(* Logix 5000 project; controller p65 vendor 1 type 14 code 85 rev 20.11; software revision 20.01; part 6 of 7 *)
(* tags used below, declared in another part *)
   DCMicroGridisInOperation : ALIAS FOR DINT00_23.8;
   DCMicroGridisSimulating : ALIAS FOR DINT00_23.10;
   Load03accountBalance : ALIAS FOR REAL00_63;
   Load03accountDepositRate : ALIAS FOR REAL00_64;
   Load03Bclose : ALIAS FOR Local:3:O.Data.7;
   Load03BcloseHILS : ALIAS FOR plc1_local_6[0].7;
   Load03BcloseProxy : ALIAS FOR DINT00_25.11;
   Load03BintReqClose : ALIAS FOR DINT00_25.12;
   Load03BisClosed : ALIAS FOR DINT00_25.13;
   Load03BisOpen : ALIAS FOR DINT00_25.14;
   Load03BreqClose : ALIAS FOR DINT00_25.15;
   Load03BreqOpen : ALIAS FOR DINT00_25.16;
   Load03commandChanged : ALIAS FOR DINT00_25.17;
   Load03commandChangedTimer : ALIAS FOR CLTIMER00_23;
   Load03current : ALIAS FOR REAL00_65;
   Load03currentHILS : ALIAS FOR plc1_local_2[7];
   Load03currentRaw : ALIAS FOR Local:2:I.Ch4Data;
   Load03deadband : ALIAS FOR REAL00_66;
   Load03depositTimer : ALIAS FOR CLTIMER00_24;
   Load03DisconnectPowerEventFail : ALIAS FOR DINT00_25.18;
   Load03DisconnectPowerEventSuccess : ALIAS FOR DINT00_25.19;
   Load03DisconnectPowerFailTimer : ALIAS FOR CLTIMER00_25;
   Load03DisconnectPowerInProcess : ALIAS FOR DINT00_25.20;
   Load03DisconnectPowerMsg : ALIAS FOR MESSAGE00_5;
   Load03DisconnectPowerSuccessTimer : ALIAS FOR CLTIMER00_26;
   Load03failedToConnect : ALIAS FOR DINT00_25.21;
   Load03failedToDisconnect : ALIAS FOR DINT00_25.22;
   Load03fundsAvailable : ALIAS FOR DINT00_25.23;
   Load03incrementToAdd : ALIAS FOR REAL00_67;
   Load03incrementToSubtract : ALIAS FOR REAL00_68;
   Load03intReqConnect : ALIAS FOR DINT00_25.24;
   Load03isConnected : ALIAS FOR DINT00_25.25;
   Load03isDisconnected : ALIAS FOR DINT00_25.26;
   Load03minBalance : ALIAS FOR REAL00_70;
   Load03minBalanceToReconnect : ALIAS FOR REAL00_71;
   Load03minTime : ALIAS FOR REAL00_72;
   Load03powerRate : ALIAS FOR REAL00_73;
   Load03powerRateMax : REAL;
   Load03PurchasePowerEventFail : ALIAS FOR DINT00_25.27;
   Load03PurchasePowerEventSuccess : ALIAS FOR DINT00_25.28;
   Load03PurchasePowerFailTimer : ALIAS FOR CLTIMER00_27;
   Load03PurchasePowerInProcess : ALIAS FOR DINT00_25.29;
   Load03PurchasePowerMsg : ALIAS FOR MESSAGE00_6;
   Load03PurchasePowerSuccessTimer : ALIAS FOR CLTIMER00_28;
   Load03reqConnect : ALIAS FOR DINT00_25.30;
   Load03reqDisconnect : ALIAS FOR DINT00_25.31;
   Load03runningOut : ALIAS FOR DINT00_26.0;
   Load03spendingRate : ALIAS FOR REAL00_74;
   Load03timeRemaining : ALIAS FOR REAL00_75;
   Load03usageTimer : ALIAS FOR CLTIMER00_29;
   Load04accountBalance : ALIAS FOR REAL00_76;
   Load04accountDepositRate : ALIAS FOR REAL00_77;
   Load04Bclose : ALIAS FOR Local:3:O.Data.8;
   Load04BcloseHILS : ALIAS FOR plc1_local_6[0].8;
   Load04BcloseProxy : ALIAS FOR DINT00_26.1;
   Load04BintReqClose : ALIAS FOR DINT00_26.2;
   Load04BisClosed : ALIAS FOR DINT00_26.3;
   Load04BisOpen : ALIAS FOR DINT00_26.4;
   Load04BreqClose : ALIAS FOR DINT00_26.5;
   Load04BreqOpen : ALIAS FOR DINT00_26.6;
   Load04commandChanged : ALIAS FOR DINT00_26.7;
   Load04commandChangedTimer : ALIAS FOR CLTIMER00_30;
   Load04current : ALIAS FOR REAL00_78;
   Load04currentHILS : ALIAS FOR plc1_local_2[8];
   Load04currentRaw : ALIAS FOR Local:2:I.Ch5Data;
   Load04deadband : ALIAS FOR REAL00_79;
   Load04depositTimer : ALIAS FOR CLTIMER00_31;
   Load04DisconnectPowerEventFail : ALIAS FOR DINT00_26.8;
   Load04DisconnectPowerEventSuccess : ALIAS FOR DINT00_26.9;
   Load04DisconnectPowerFailTimer : ALIAS FOR CLTIMER00_32;
   Load04DisconnectPowerInProcess : ALIAS FOR DINT00_26.10;
   Load04DisconnectPowerMsg : ALIAS FOR MESSAGE00_7;
   Load04DisconnectPowerSuccessTimer : ALIAS FOR CLTIMER00_33;
   Load04failedToConnect : ALIAS FOR DINT00_26.11;
   Load04failedToDisconnect : ALIAS FOR DINT00_26.12;
   Load04fundsAvailable : ALIAS FOR DINT00_26.13;
   Load04incrementToAdd : ALIAS FOR REAL00_80;
   Load04incrementToSubtract : ALIAS FOR REAL00_81;
   Load04intReqConnect : ALIAS FOR DINT00_26.14;
   Load04isConnected : ALIAS FOR DINT00_26.15;
   Load04isDisconnected : ALIAS FOR DINT00_26.16;
   Load04minBalance : ALIAS FOR REAL00_83;
   Load04minBalanceToReconnect : ALIAS FOR REAL00_84;
   Load04minTime : ALIAS FOR REAL00_85;
   Load04powerRate : ALIAS FOR REAL00_86;
   Load04powerRateMax : REAL;
   Load04PurchasePowerEventFail : ALIAS FOR DINT00_26.17;
   Load04PurchasePowerEventSuccess : ALIAS FOR DINT00_26.18;
   Load04PurchasePowerFailTimer : ALIAS FOR CLTIMER00_34;
   Load04PurchasePowerInProcess : ALIAS FOR DINT00_26.19;
   Load04PurchasePowerMsg : ALIAS FOR MESSAGE00_8;
   Load04PurchasePowerSuccessTimer : ALIAS FOR CLTIMER00_35;
   Load04reqConnect : ALIAS FOR DINT00_26.20;
   Load04reqDisconnect : ALIAS FOR DINT00_26.21;
   Load04runningOut : ALIAS FOR DINT00_26.22;
   Load04spendingRate : ALIAS FOR REAL00_87;
   Load04timeRemaining : ALIAS FOR REAL00_88;
   Load04usageTimer : ALIAS FOR CLTIMER00_36;
   Load05accountBalance : ALIAS FOR REAL00_89;
   Load05accountDepositRate : ALIAS FOR REAL00_90;
   Load05Bclose : ALIAS FOR Local:3:O.Data.9;
   Load05BcloseHILS : ALIAS FOR plc1_local_6[0].9;
   Load05BcloseProxy : ALIAS FOR DINT00_26.23;
   Load05BintReqClose : ALIAS FOR DINT00_26.24;
   Load05BisClosed : ALIAS FOR DINT00_26.25;
   Load05BisOpen : ALIAS FOR DINT00_26.26;
   Load05BreqClose : ALIAS FOR DINT00_26.27;
   Load05BreqOpen : ALIAS FOR DINT00_26.28;
   Load05commandChanged : ALIAS FOR DINT00_26.29;
   Load05commandChangedTimer : ALIAS FOR CLTIMER00_37;
   Load05current : ALIAS FOR REAL00_91;
   Load05currentHILS : ALIAS FOR plc1_local_2[9];
   Load05currentRaw : ALIAS FOR Local:2:I.Ch6Data;
   Load05deadband : ALIAS FOR REAL00_92;
   Load05depositTimer : ALIAS FOR CLTIMER00_38;
   Load05DisconnectPowerEventFail : ALIAS FOR DINT00_26.30;
   Load05DisconnectPowerEventSuccess : ALIAS FOR DINT00_26.31;
   Load05DisconnectPowerFailTimer : ALIAS FOR CLTIMER00_39;
   Load05DisconnectPowerInProcess : ALIAS FOR DINT00_27.0;
   Load05DisconnectPowerMsg : ALIAS FOR MESSAGE00_9;
   Load05DisconnectPowerSuccessTimer : ALIAS FOR CLTIMER00_40;
   Load05failedToConnect : ALIAS FOR DINT00_27.1;
   Load05failedToDisconnect : ALIAS FOR DINT00_27.2;
   Load05fundsAvailable : ALIAS FOR DINT00_27.3;
   Load05incrementToAdd : ALIAS FOR REAL00_93;
   Load05incrementToSubtract : ALIAS FOR REAL00_94;
   Load05intReqConnect : ALIAS FOR DINT00_27.4;
   Load05isConnected : ALIAS FOR DINT00_27.5;
   Load05isDisconnected : ALIAS FOR DINT00_27.6;
   Load05minBalance : ALIAS FOR REAL00_96;
   Load05minBalanceToReconnect : ALIAS FOR REAL00_97;
   Load05minTime : ALIAS FOR REAL00_98;
   Load05powerRate : ALIAS FOR REAL00_99;
   Load05powerRateMax : REAL;
   Load05PurchasePowerEventFail : ALIAS FOR DINT00_27.7;
   Load05PurchasePowerEventSuccess : ALIAS FOR DINT00_27.8;
   Load05PurchasePowerFailTimer : ALIAS FOR CLTIMER00_41;
   Load05PurchasePowerInProcess : ALIAS FOR DINT00_27.9;
   Load05PurchasePowerMsg : ALIAS FOR MESSAGE00_10;
   Load05PurchasePowerSuccessTimer : ALIAS FOR CLTIMER00_42;
   Load05reqConnect : ALIAS FOR DINT00_27.10;
   Load05reqDisconnect : ALIAS FOR DINT00_27.11;
   Load05runningOut : ALIAS FOR DINT00_27.12;
   Load05spendingRate : ALIAS FOR REAL00_100;
   Load05timeRemaining : ALIAS FOR REAL00_101;
   Load05usageTimer : ALIAS FOR CLTIMER00_43;
   LoadslowVoltage : ALIAS FOR DINT00_27.23;
   UsingAgents : BOOL;

PROGRAM Load03   (* main routine Load03 *)

ROUTINE Load03   (* ladder *)
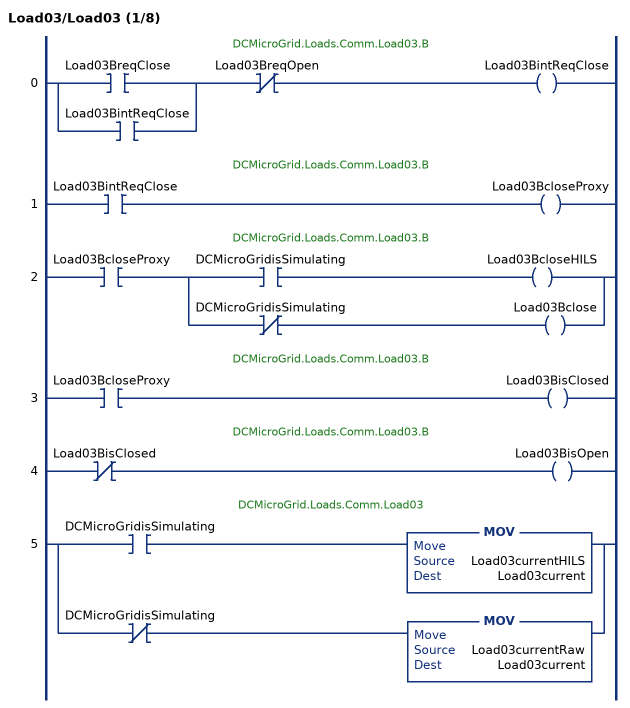
   // DCMicroGrid.Loads.Comm.Load03.B
   0: [XIC(Load03BreqClose) ,XIC(Load03BintReqClose) ]XIO(Load03BreqOpen)OTE(Load03BintReqClose);
   // DCMicroGrid.Loads.Comm.Load03.B
   1: XIC(Load03BintReqClose)OTE(Load03BcloseProxy);
   // DCMicroGrid.Loads.Comm.Load03.B
   2: XIC(Load03BcloseProxy)[XIC(DCMicroGridisSimulating) OTE(Load03BcloseHILS) ,XIO(DCMicroGridisSimulating) OTE(Load03Bclose) ];
   // DCMicroGrid.Loads.Comm.Load03.B
   3: XIC(Load03BcloseProxy)OTE(Load03BisClosed);
   // DCMicroGrid.Loads.Comm.Load03.B
   4: XIO(Load03BisClosed)OTE(Load03BisOpen);
   // DCMicroGrid.Loads.Comm.Load03
   5: [XIC(DCMicroGridisSimulating) MOV(Load03currentHILS,Load03current) ,XIO(DCMicroGridisSimulating) MOV(Load03currentRaw,Load03current) ];
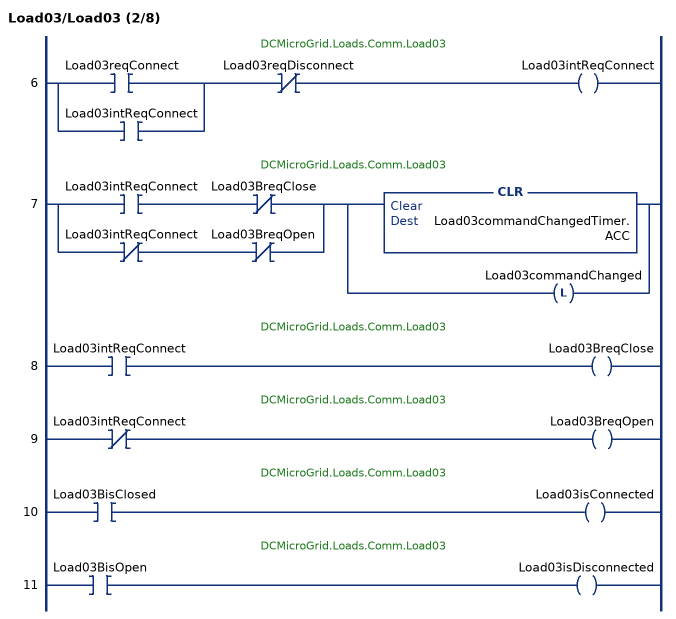
   // DCMicroGrid.Loads.Comm.Load03
   6: [XIC(Load03reqConnect) ,XIC(Load03intReqConnect) ]XIO(Load03reqDisconnect)OTE(Load03intReqConnect);
   // DCMicroGrid.Loads.Comm.Load03
   7: [XIC(Load03intReqConnect) XIO(Load03BreqClose) ,XIO(Load03intReqConnect) XIO(Load03BreqOpen) ][CLR(Load03commandChangedTimer.ACC) ,OTL(Load03commandChanged) ];
   // DCMicroGrid.Loads.Comm.Load03
   8: XIC(Load03intReqConnect)OTE(Load03BreqClose);
   // DCMicroGrid.Loads.Comm.Load03
   9: XIO(Load03intReqConnect)OTE(Load03BreqOpen);
   // DCMicroGrid.Loads.Comm.Load03
   10: XIC(Load03BisClosed)OTE(Load03isConnected);
   // DCMicroGrid.Loads.Comm.Load03
   11: XIC(Load03BisOpen)OTE(Load03isDisconnected);
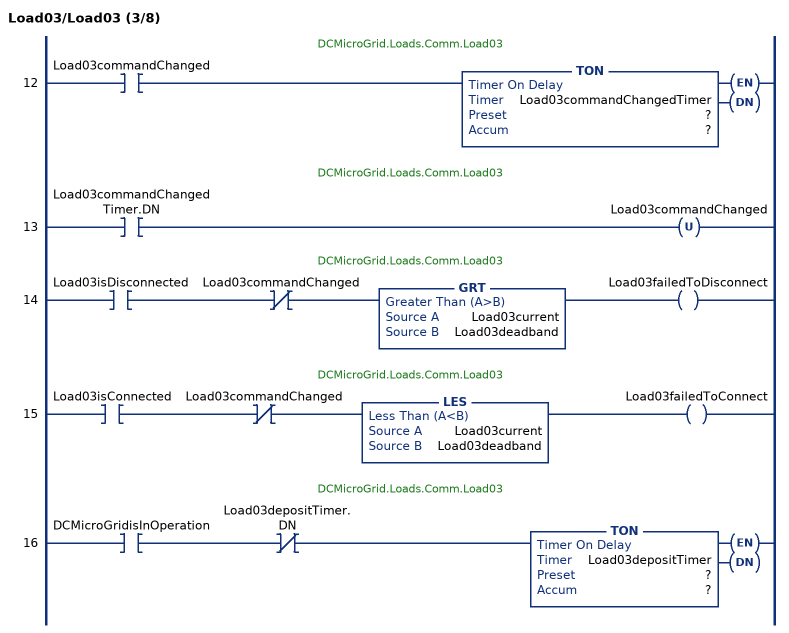
   // DCMicroGrid.Loads.Comm.Load03
   12: XIC(Load03commandChanged)TON(Load03commandChangedTimer,?,?);
   // DCMicroGrid.Loads.Comm.Load03
   13: XIC(Load03commandChangedTimer.DN)OTU(Load03commandChanged);
   // DCMicroGrid.Loads.Comm.Load03
   14: XIC(Load03isDisconnected)XIO(Load03commandChanged)GRT(Load03current,Load03deadband)OTE(Load03failedToDisconnect);
   // DCMicroGrid.Loads.Comm.Load03
   15: XIC(Load03isConnected)XIO(Load03commandChanged)LES(Load03current,Load03deadband)OTE(Load03failedToConnect);
   // DCMicroGrid.Loads.Comm.Load03
   16: XIC(DCMicroGridisInOperation)XIO(Load03depositTimer.DN)TON(Load03depositTimer,?,?);
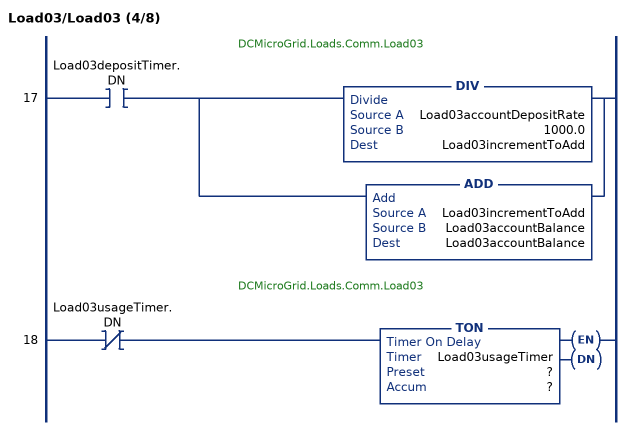
   // DCMicroGrid.Loads.Comm.Load03
   17: XIC(Load03depositTimer.DN)[DIV(Load03accountDepositRate,1000.0,Load03incrementToAdd) ,ADD(Load03incrementToAdd,Load03accountBalance,Load03accountBalance) ];
   // DCMicroGrid.Loads.Comm.Load03
   18: XIO(Load03usageTimer.DN)TON(Load03usageTimer,?,?);
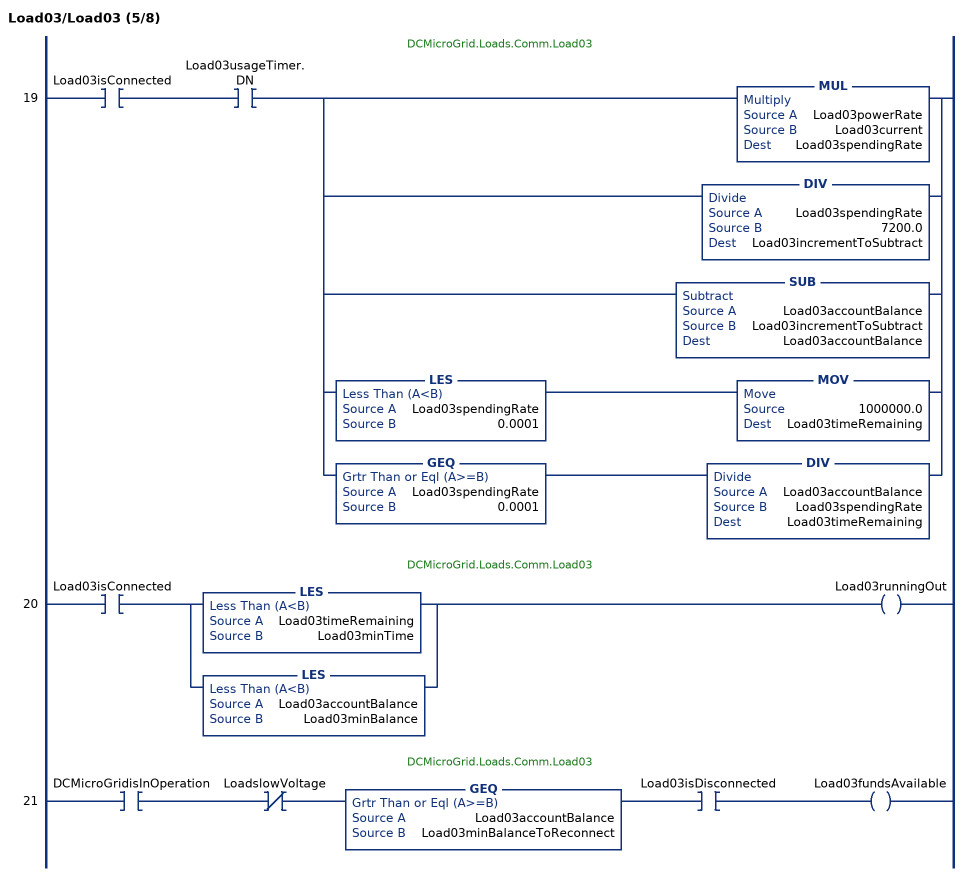
   // DCMicroGrid.Loads.Comm.Load03
   19: XIC(Load03isConnected)XIC(Load03usageTimer.DN)[MUL(Load03powerRate,Load03current,Load03spendingRate) ,DIV(Load03spendingRate,7200.0,Load03incrementToSubtract) ,SUB(Load03accountBalance,Load03incrementToSubtract,Load03accountBalance) ,[LES(Load03spendingRate,0.0001) MOV(1000000.0,Load03timeRemaining) ,GEQ(Load03spendingRate,0.0001) DIV(Load03accountBalance,Load03spendingRate,Load03timeRemaining) ] ];
   // DCMicroGrid.Loads.Comm.Load03
   20: XIC(Load03isConnected)[LES(Load03timeRemaining,Load03minTime) ,LES(Load03accountBalance,Load03minBalance) ]OTE(Load03runningOut);
   // DCMicroGrid.Loads.Comm.Load03
   21: XIC(DCMicroGridisInOperation)XIO(LoadslowVoltage)GEQ(Load03accountBalance,Load03minBalanceToReconnect)XIC(Load03isDisconnected)OTE(Load03fundsAvailable);
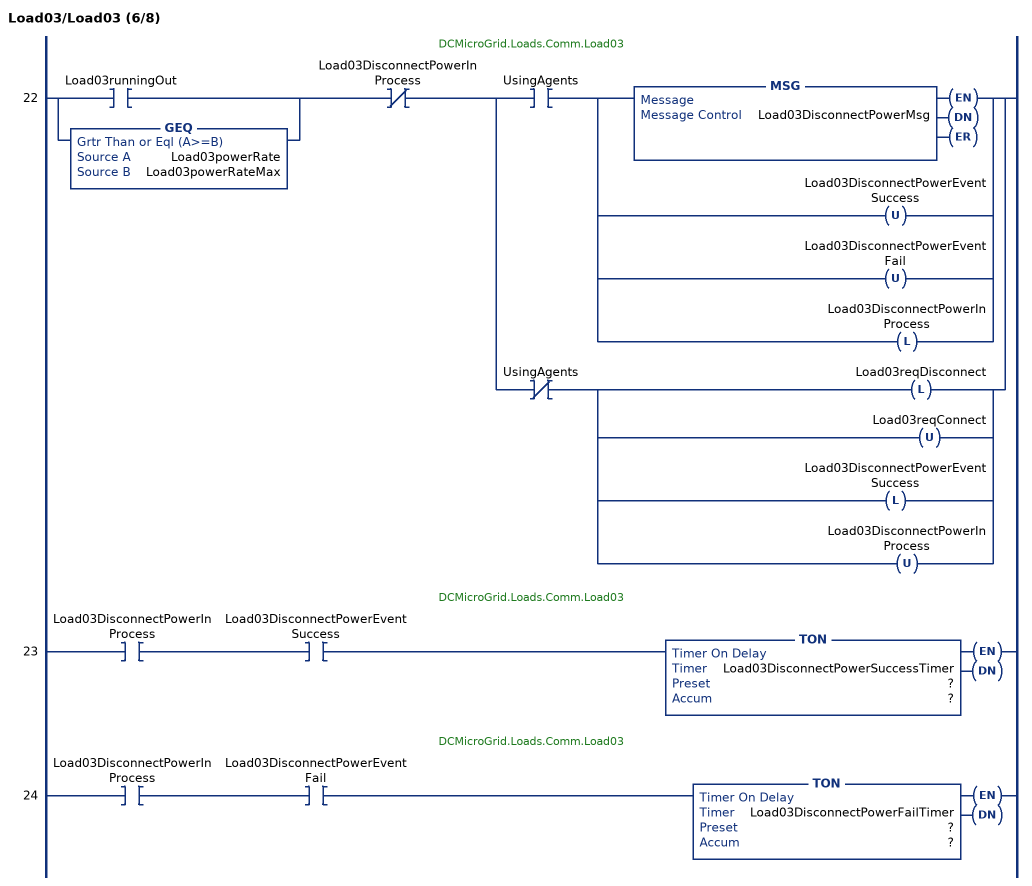
   // DCMicroGrid.Loads.Comm.Load03
   22: [XIC(Load03runningOut) ,GEQ(Load03powerRate,Load03powerRateMax) ]XIO(Load03DisconnectPowerInProcess)[XIC(UsingAgents) [MSG(Load03DisconnectPowerMsg) ,OTU(Load03DisconnectPowerEventSuccess) ,OTU(Load03DisconnectPowerEventFail) ,OTL(Load03DisconnectPowerInProcess) ] ,XIO(UsingAgents) [OTL(Load03reqDisconnect) ,OTU(Load03reqConnect) ,OTL(Load03DisconnectPowerEventSuccess) ,OTU(Load03DisconnectPowerInProcess) ] ];
   // DCMicroGrid.Loads.Comm.Load03
   23: XIC(Load03DisconnectPowerInProcess)XIC(Load03DisconnectPowerEventSuccess)TON(Load03DisconnectPowerSuccessTimer,?,?);
   // DCMicroGrid.Loads.Comm.Load03
   24: XIC(Load03DisconnectPowerInProcess)XIC(Load03DisconnectPowerEventFail)TON(Load03DisconnectPowerFailTimer,?,?);
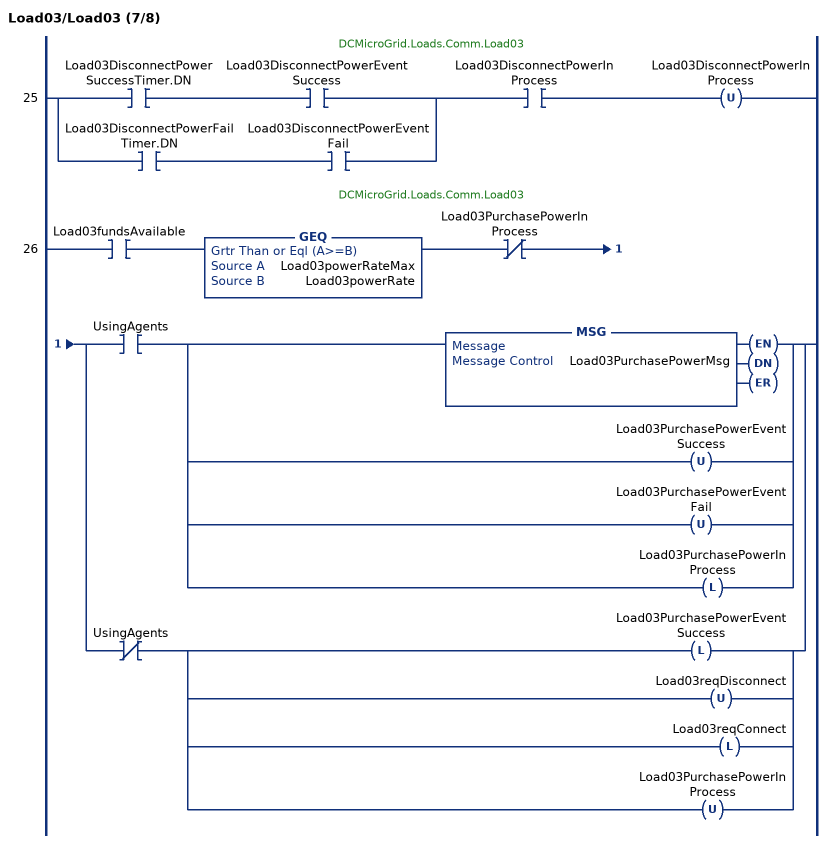
   // DCMicroGrid.Loads.Comm.Load03
   25: [XIC(Load03DisconnectPowerSuccessTimer.DN) XIC(Load03DisconnectPowerEventSuccess) ,XIC(Load03DisconnectPowerFailTimer.DN) XIC(Load03DisconnectPowerEventFail) ]XIC(Load03DisconnectPowerInProcess)OTU(Load03DisconnectPowerInProcess);
   // DCMicroGrid.Loads.Comm.Load03
   26: XIC(Load03fundsAvailable)GEQ(Load03powerRateMax,Load03powerRate)XIO(Load03PurchasePowerInProcess)[XIC(UsingAgents) [MSG(Load03PurchasePowerMsg) ,OTU(Load03PurchasePowerEventSuccess) ,OTU(Load03PurchasePowerEventFail) ,OTL(Load03PurchasePowerInProcess) ] ,XIO(UsingAgents) [OTL(Load03PurchasePowerEventSuccess) ,OTU(Load03reqDisconnect) ,OTL(Load03reqConnect) ,OTU(Load03PurchasePowerInProcess) ] ];
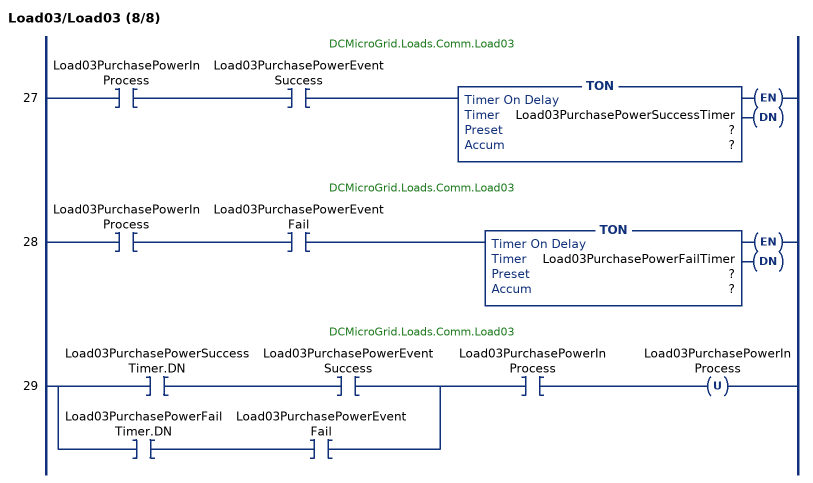
   // DCMicroGrid.Loads.Comm.Load03
   27: XIC(Load03PurchasePowerInProcess)XIC(Load03PurchasePowerEventSuccess)TON(Load03PurchasePowerSuccessTimer,?,?);
   // DCMicroGrid.Loads.Comm.Load03
   28: XIC(Load03PurchasePowerInProcess)XIC(Load03PurchasePowerEventFail)TON(Load03PurchasePowerFailTimer,?,?);
   // DCMicroGrid.Loads.Comm.Load03
   29: [XIC(Load03PurchasePowerSuccessTimer.DN) XIC(Load03PurchasePowerEventSuccess) ,XIC(Load03PurchasePowerFailTimer.DN) XIC(Load03PurchasePowerEventFail) ]XIC(Load03PurchasePowerInProcess)OTU(Load03PurchasePowerInProcess);
END_ROUTINE
END_PROGRAM

PROGRAM Load04   (* main routine Load04 *)

ROUTINE Load04   (* ladder *)
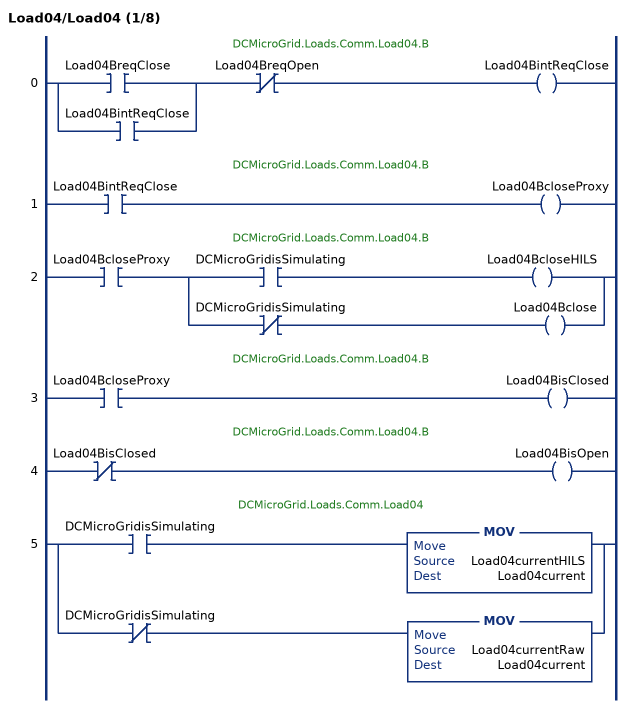
   // DCMicroGrid.Loads.Comm.Load04.B
   0: [XIC(Load04BreqClose) ,XIC(Load04BintReqClose) ]XIO(Load04BreqOpen)OTE(Load04BintReqClose);
   // DCMicroGrid.Loads.Comm.Load04.B
   1: XIC(Load04BintReqClose)OTE(Load04BcloseProxy);
   // DCMicroGrid.Loads.Comm.Load04.B
   2: XIC(Load04BcloseProxy)[XIC(DCMicroGridisSimulating) OTE(Load04BcloseHILS) ,XIO(DCMicroGridisSimulating) OTE(Load04Bclose) ];
   // DCMicroGrid.Loads.Comm.Load04.B
   3: XIC(Load04BcloseProxy)OTE(Load04BisClosed);
   // DCMicroGrid.Loads.Comm.Load04.B
   4: XIO(Load04BisClosed)OTE(Load04BisOpen);
   // DCMicroGrid.Loads.Comm.Load04
   5: [XIC(DCMicroGridisSimulating) MOV(Load04currentHILS,Load04current) ,XIO(DCMicroGridisSimulating) MOV(Load04currentRaw,Load04current) ];
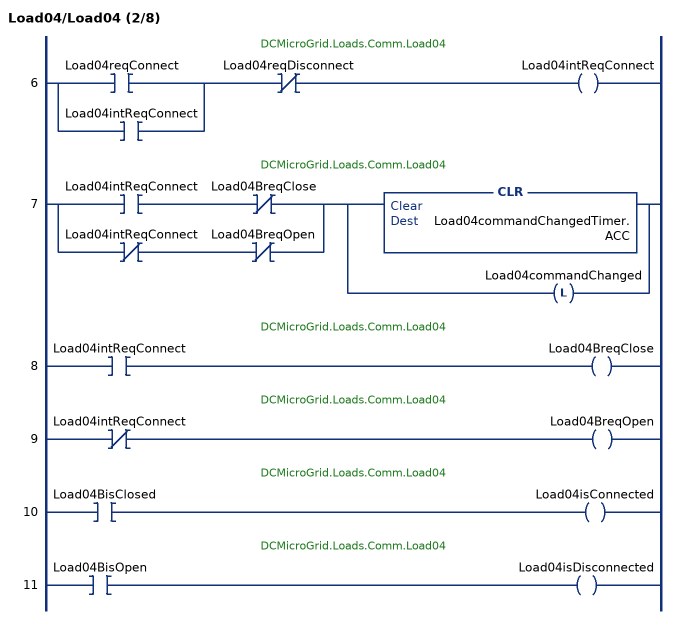
   // DCMicroGrid.Loads.Comm.Load04
   6: [XIC(Load04reqConnect) ,XIC(Load04intReqConnect) ]XIO(Load04reqDisconnect)OTE(Load04intReqConnect);
   // DCMicroGrid.Loads.Comm.Load04
   7: [XIC(Load04intReqConnect) XIO(Load04BreqClose) ,XIO(Load04intReqConnect) XIO(Load04BreqOpen) ][CLR(Load04commandChangedTimer.ACC) ,OTL(Load04commandChanged) ];
   // DCMicroGrid.Loads.Comm.Load04
   8: XIC(Load04intReqConnect)OTE(Load04BreqClose);
   // DCMicroGrid.Loads.Comm.Load04
   9: XIO(Load04intReqConnect)OTE(Load04BreqOpen);
   // DCMicroGrid.Loads.Comm.Load04
   10: XIC(Load04BisClosed)OTE(Load04isConnected);
   // DCMicroGrid.Loads.Comm.Load04
   11: XIC(Load04BisOpen)OTE(Load04isDisconnected);
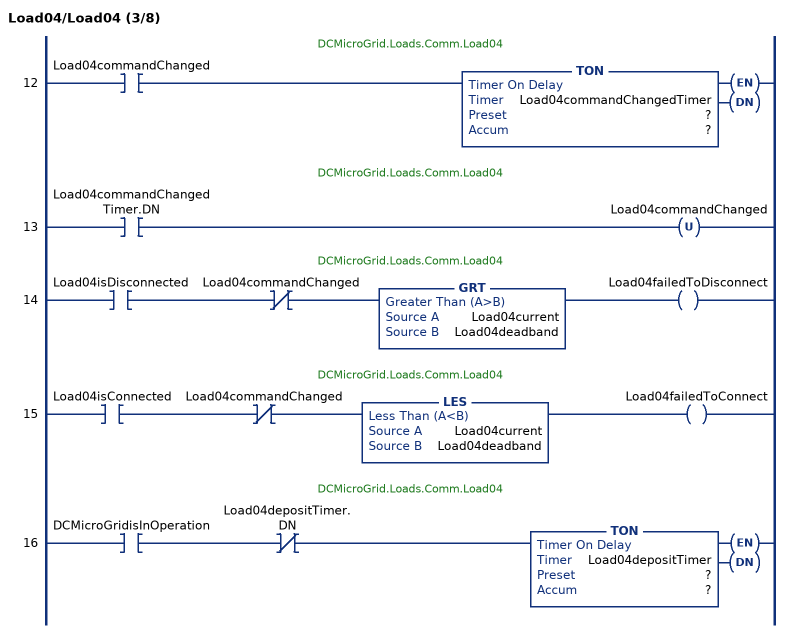
   // DCMicroGrid.Loads.Comm.Load04
   12: XIC(Load04commandChanged)TON(Load04commandChangedTimer,?,?);
   // DCMicroGrid.Loads.Comm.Load04
   13: XIC(Load04commandChangedTimer.DN)OTU(Load04commandChanged);
   // DCMicroGrid.Loads.Comm.Load04
   14: XIC(Load04isDisconnected)XIO(Load04commandChanged)GRT(Load04current,Load04deadband)OTE(Load04failedToDisconnect);
   // DCMicroGrid.Loads.Comm.Load04
   15: XIC(Load04isConnected)XIO(Load04commandChanged)LES(Load04current,Load04deadband)OTE(Load04failedToConnect);
   // DCMicroGrid.Loads.Comm.Load04
   16: XIC(DCMicroGridisInOperation)XIO(Load04depositTimer.DN)TON(Load04depositTimer,?,?);
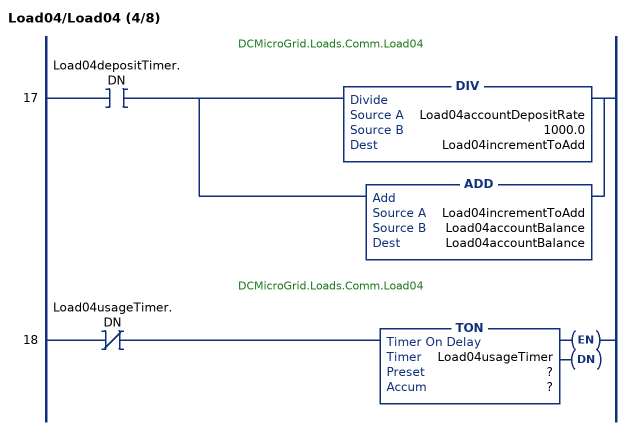
   // DCMicroGrid.Loads.Comm.Load04
   17: XIC(Load04depositTimer.DN)[DIV(Load04accountDepositRate,1000.0,Load04incrementToAdd) ,ADD(Load04incrementToAdd,Load04accountBalance,Load04accountBalance) ];
   // DCMicroGrid.Loads.Comm.Load04
   18: XIO(Load04usageTimer.DN)TON(Load04usageTimer,?,?);
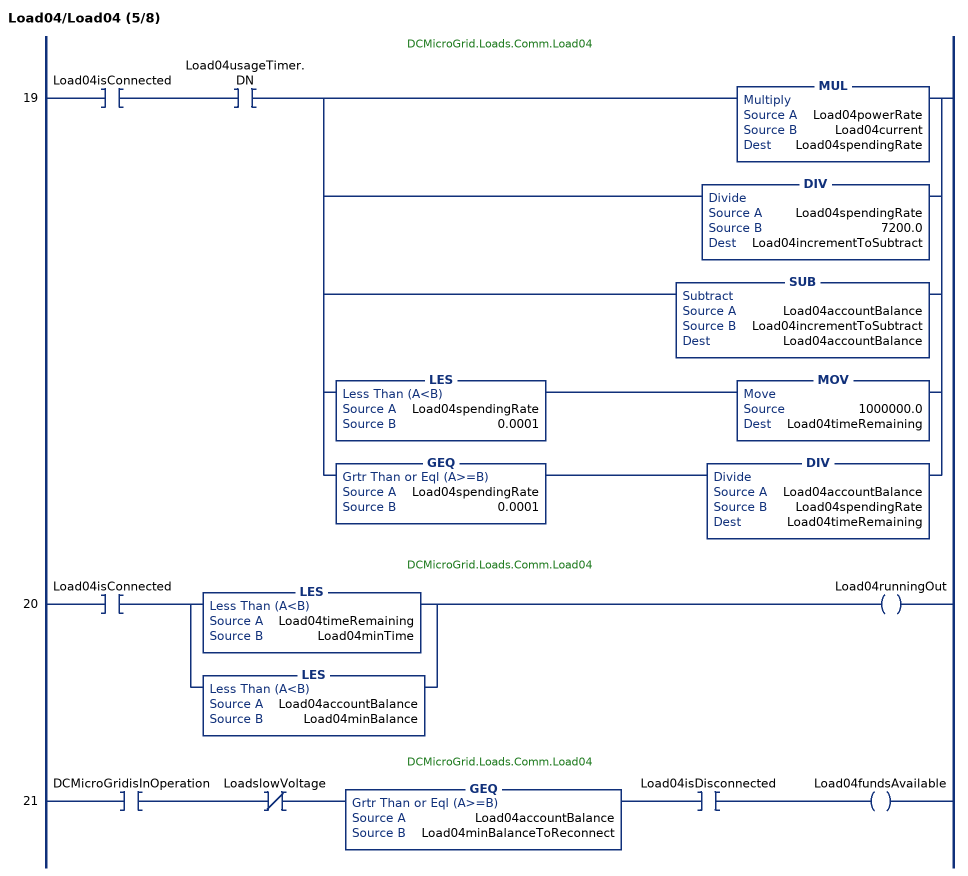
   // DCMicroGrid.Loads.Comm.Load04
   19: XIC(Load04isConnected)XIC(Load04usageTimer.DN)[MUL(Load04powerRate,Load04current,Load04spendingRate) ,DIV(Load04spendingRate,7200.0,Load04incrementToSubtract) ,SUB(Load04accountBalance,Load04incrementToSubtract,Load04accountBalance) ,[LES(Load04spendingRate,0.0001) MOV(1000000.0,Load04timeRemaining) ,GEQ(Load04spendingRate,0.0001) DIV(Load04accountBalance,Load04spendingRate,Load04timeRemaining) ] ];
   // DCMicroGrid.Loads.Comm.Load04
   20: XIC(Load04isConnected)[LES(Load04timeRemaining,Load04minTime) ,LES(Load04accountBalance,Load04minBalance) ]OTE(Load04runningOut);
   // DCMicroGrid.Loads.Comm.Load04
   21: XIC(DCMicroGridisInOperation)XIO(LoadslowVoltage)GEQ(Load04accountBalance,Load04minBalanceToReconnect)XIC(Load04isDisconnected)OTE(Load04fundsAvailable);
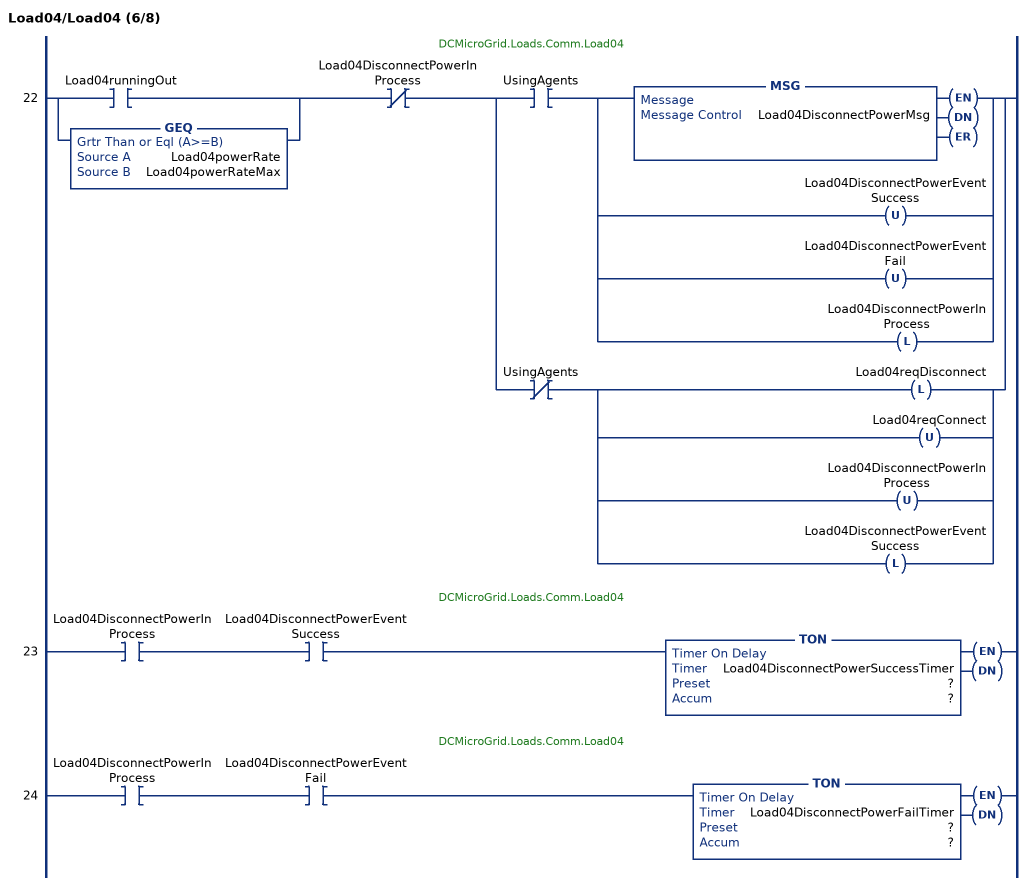
   // DCMicroGrid.Loads.Comm.Load04
   22: [XIC(Load04runningOut) ,GEQ(Load04powerRate,Load04powerRateMax) ]XIO(Load04DisconnectPowerInProcess)[XIC(UsingAgents) [MSG(Load04DisconnectPowerMsg) ,OTU(Load04DisconnectPowerEventSuccess) ,OTU(Load04DisconnectPowerEventFail) ,OTL(Load04DisconnectPowerInProcess) ] ,XIO(UsingAgents) [OTL(Load04reqDisconnect) ,OTU(Load04reqConnect) ,OTU(Load04DisconnectPowerInProcess) ,OTL(Load04DisconnectPowerEventSuccess) ] ];
   // DCMicroGrid.Loads.Comm.Load04
   23: XIC(Load04DisconnectPowerInProcess)XIC(Load04DisconnectPowerEventSuccess)TON(Load04DisconnectPowerSuccessTimer,?,?);
   // DCMicroGrid.Loads.Comm.Load04
   24: XIC(Load04DisconnectPowerInProcess)XIC(Load04DisconnectPowerEventFail)TON(Load04DisconnectPowerFailTimer,?,?);
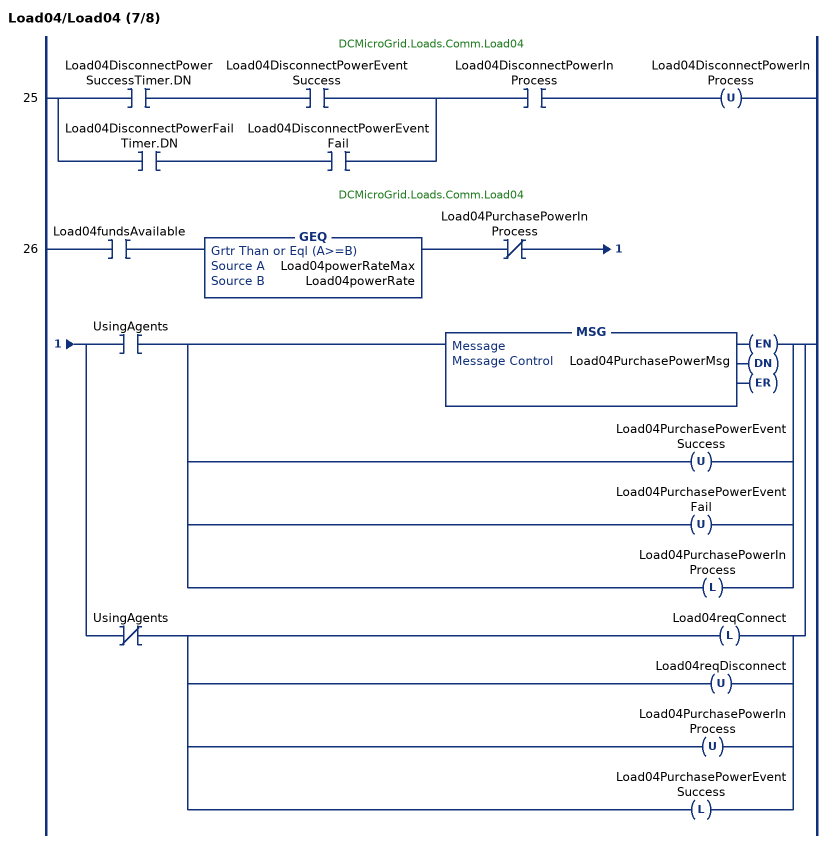
   // DCMicroGrid.Loads.Comm.Load04
   25: [XIC(Load04DisconnectPowerSuccessTimer.DN) XIC(Load04DisconnectPowerEventSuccess) ,XIC(Load04DisconnectPowerFailTimer.DN) XIC(Load04DisconnectPowerEventFail) ]XIC(Load04DisconnectPowerInProcess)OTU(Load04DisconnectPowerInProcess);
   // DCMicroGrid.Loads.Comm.Load04
   26: XIC(Load04fundsAvailable)GEQ(Load04powerRateMax,Load04powerRate)XIO(Load04PurchasePowerInProcess)[XIC(UsingAgents) [MSG(Load04PurchasePowerMsg) ,OTU(Load04PurchasePowerEventSuccess) ,OTU(Load04PurchasePowerEventFail) ,OTL(Load04PurchasePowerInProcess) ] ,XIO(UsingAgents) [OTL(Load04reqConnect) ,OTU(Load04reqDisconnect) ,OTU(Load04PurchasePowerInProcess) ,OTL(Load04PurchasePowerEventSuccess) ] ];
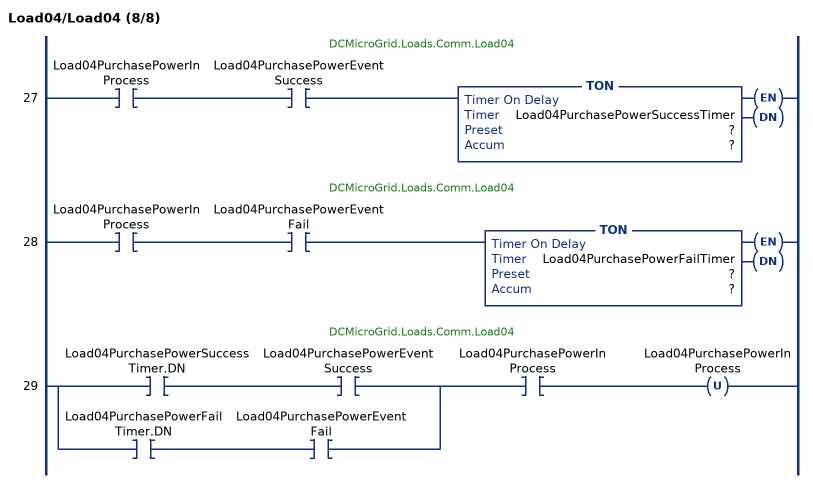
   // DCMicroGrid.Loads.Comm.Load04
   27: XIC(Load04PurchasePowerInProcess)XIC(Load04PurchasePowerEventSuccess)TON(Load04PurchasePowerSuccessTimer,?,?);
   // DCMicroGrid.Loads.Comm.Load04
   28: XIC(Load04PurchasePowerInProcess)XIC(Load04PurchasePowerEventFail)TON(Load04PurchasePowerFailTimer,?,?);
   // DCMicroGrid.Loads.Comm.Load04
   29: [XIC(Load04PurchasePowerSuccessTimer.DN) XIC(Load04PurchasePowerEventSuccess) ,XIC(Load04PurchasePowerFailTimer.DN) XIC(Load04PurchasePowerEventFail) ]XIC(Load04PurchasePowerInProcess)OTU(Load04PurchasePowerInProcess);
END_ROUTINE
END_PROGRAM

PROGRAM Load05   (* main routine Load05 *)

ROUTINE Load05   (* ladder *)
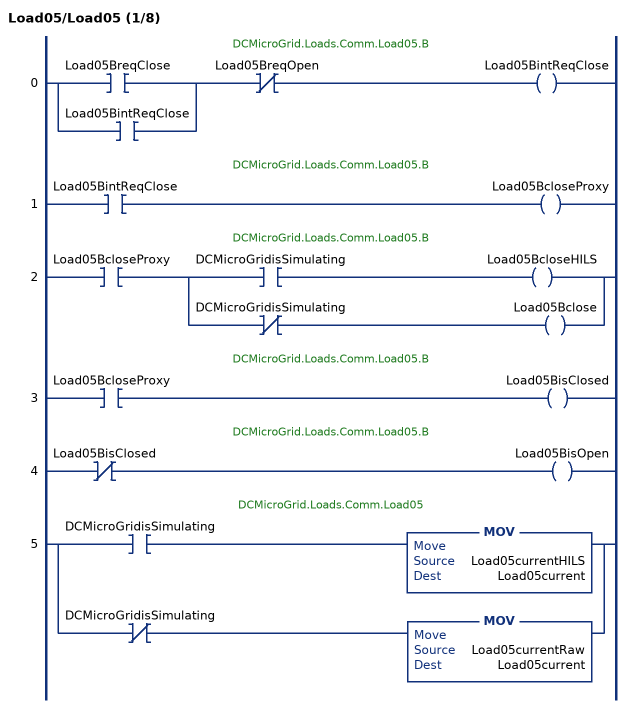
   // DCMicroGrid.Loads.Comm.Load05.B
   0: [XIC(Load05BreqClose) ,XIC(Load05BintReqClose) ]XIO(Load05BreqOpen)OTE(Load05BintReqClose);
   // DCMicroGrid.Loads.Comm.Load05.B
   1: XIC(Load05BintReqClose)OTE(Load05BcloseProxy);
   // DCMicroGrid.Loads.Comm.Load05.B
   2: XIC(Load05BcloseProxy)[XIC(DCMicroGridisSimulating) OTE(Load05BcloseHILS) ,XIO(DCMicroGridisSimulating) OTE(Load05Bclose) ];
   // DCMicroGrid.Loads.Comm.Load05.B
   3: XIC(Load05BcloseProxy)OTE(Load05BisClosed);
   // DCMicroGrid.Loads.Comm.Load05.B
   4: XIO(Load05BisClosed)OTE(Load05BisOpen);
   // DCMicroGrid.Loads.Comm.Load05
   5: [XIC(DCMicroGridisSimulating) MOV(Load05currentHILS,Load05current) ,XIO(DCMicroGridisSimulating) MOV(Load05currentRaw,Load05current) ];
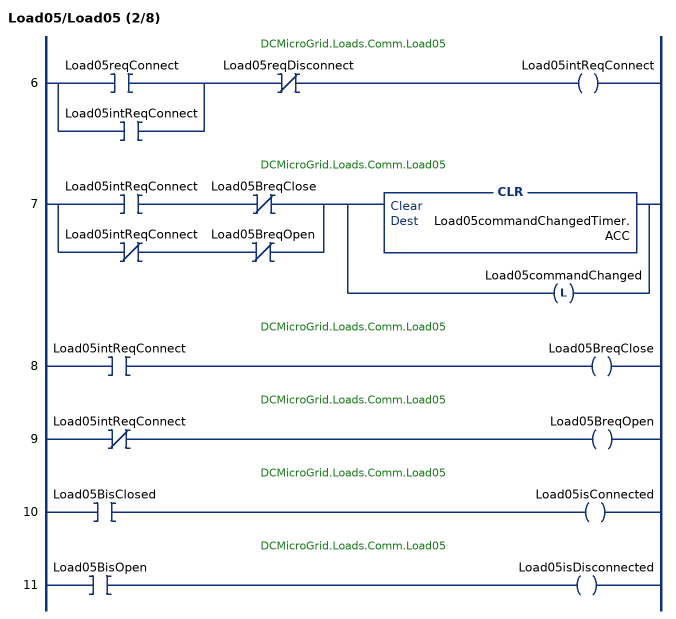
   // DCMicroGrid.Loads.Comm.Load05
   6: [XIC(Load05reqConnect) ,XIC(Load05intReqConnect) ]XIO(Load05reqDisconnect)OTE(Load05intReqConnect);
   // DCMicroGrid.Loads.Comm.Load05
   7: [XIC(Load05intReqConnect) XIO(Load05BreqClose) ,XIO(Load05intReqConnect) XIO(Load05BreqOpen) ][CLR(Load05commandChangedTimer.ACC) ,OTL(Load05commandChanged) ];
   // DCMicroGrid.Loads.Comm.Load05
   8: XIC(Load05intReqConnect)OTE(Load05BreqClose);
   // DCMicroGrid.Loads.Comm.Load05
   9: XIO(Load05intReqConnect)OTE(Load05BreqOpen);
   // DCMicroGrid.Loads.Comm.Load05
   10: XIC(Load05BisClosed)OTE(Load05isConnected);
   // DCMicroGrid.Loads.Comm.Load05
   11: XIC(Load05BisOpen)OTE(Load05isDisconnected);
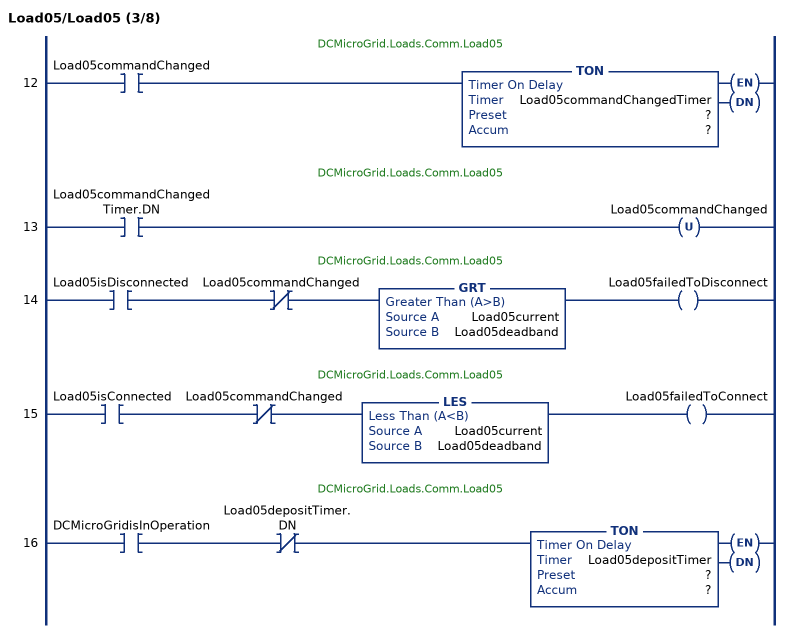
   // DCMicroGrid.Loads.Comm.Load05
   12: XIC(Load05commandChanged)TON(Load05commandChangedTimer,?,?);
   // DCMicroGrid.Loads.Comm.Load05
   13: XIC(Load05commandChangedTimer.DN)OTU(Load05commandChanged);
   // DCMicroGrid.Loads.Comm.Load05
   14: XIC(Load05isDisconnected)XIO(Load05commandChanged)GRT(Load05current,Load05deadband)OTE(Load05failedToDisconnect);
   // DCMicroGrid.Loads.Comm.Load05
   15: XIC(Load05isConnected)XIO(Load05commandChanged)LES(Load05current,Load05deadband)OTE(Load05failedToConnect);
   // DCMicroGrid.Loads.Comm.Load05
   16: XIC(DCMicroGridisInOperation)XIO(Load05depositTimer.DN)TON(Load05depositTimer,?,?);
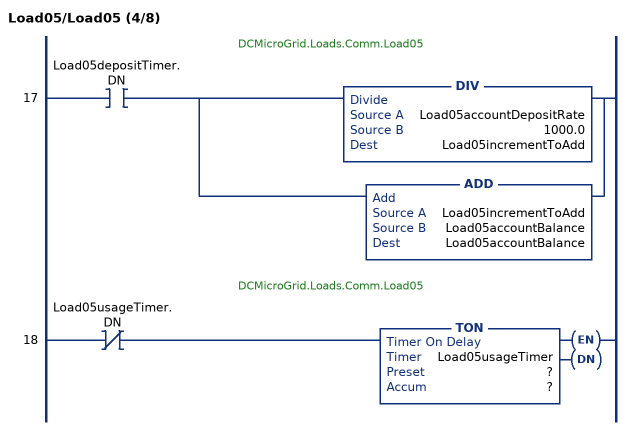
   // DCMicroGrid.Loads.Comm.Load05
   17: XIC(Load05depositTimer.DN)[DIV(Load05accountDepositRate,1000.0,Load05incrementToAdd) ,ADD(Load05incrementToAdd,Load05accountBalance,Load05accountBalance) ];
   // DCMicroGrid.Loads.Comm.Load05
   18: XIO(Load05usageTimer.DN)TON(Load05usageTimer,?,?);
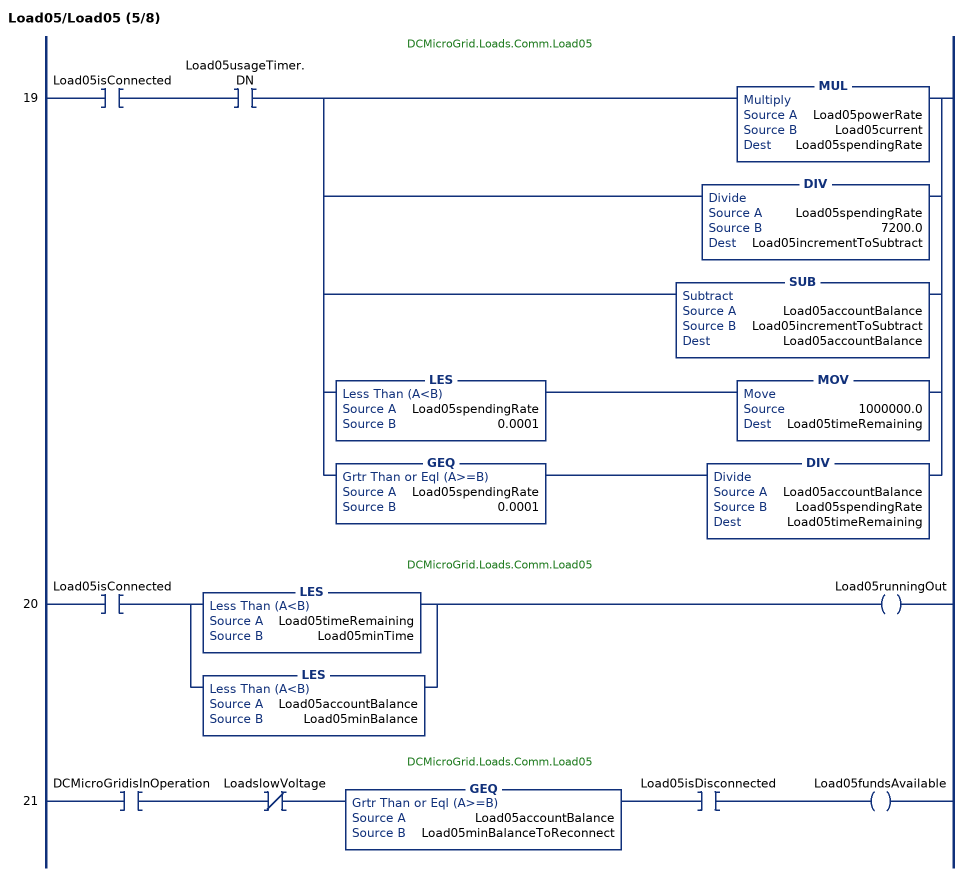
   // DCMicroGrid.Loads.Comm.Load05
   19: XIC(Load05isConnected)XIC(Load05usageTimer.DN)[MUL(Load05powerRate,Load05current,Load05spendingRate) ,DIV(Load05spendingRate,7200.0,Load05incrementToSubtract) ,SUB(Load05accountBalance,Load05incrementToSubtract,Load05accountBalance) ,[LES(Load05spendingRate,0.0001) MOV(1000000.0,Load05timeRemaining) ,GEQ(Load05spendingRate,0.0001) DIV(Load05accountBalance,Load05spendingRate,Load05timeRemaining) ] ];
   // DCMicroGrid.Loads.Comm.Load05
   20: XIC(Load05isConnected)[LES(Load05timeRemaining,Load05minTime) ,LES(Load05accountBalance,Load05minBalance) ]OTE(Load05runningOut);
   // DCMicroGrid.Loads.Comm.Load05
   21: XIC(DCMicroGridisInOperation)XIO(LoadslowVoltage)GEQ(Load05accountBalance,Load05minBalanceToReconnect)XIC(Load05isDisconnected)OTE(Load05fundsAvailable);
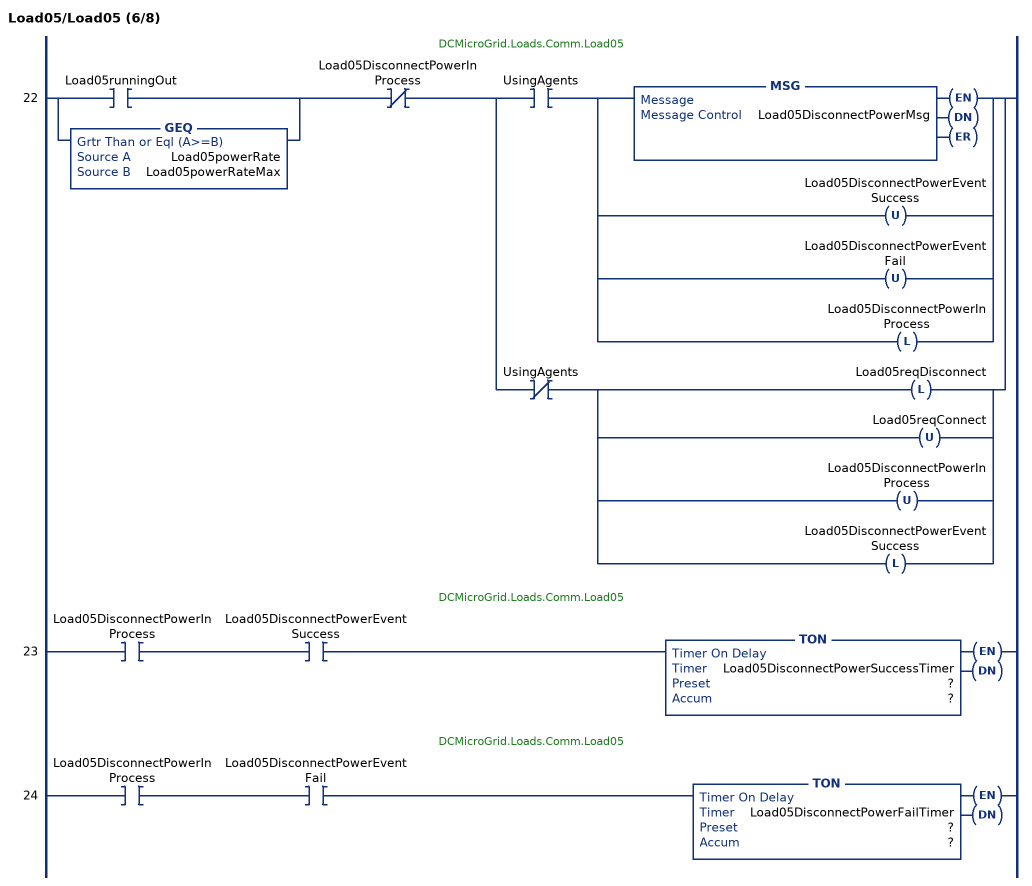
   // DCMicroGrid.Loads.Comm.Load05
   22: [XIC(Load05runningOut) ,GEQ(Load05powerRate,Load05powerRateMax) ]XIO(Load05DisconnectPowerInProcess)[XIC(UsingAgents) [MSG(Load05DisconnectPowerMsg) ,OTU(Load05DisconnectPowerEventSuccess) ,OTU(Load05DisconnectPowerEventFail) ,OTL(Load05DisconnectPowerInProcess) ] ,XIO(UsingAgents) [OTL(Load05reqDisconnect) ,OTU(Load05reqConnect) ,OTU(Load05DisconnectPowerInProcess) ,OTL(Load05DisconnectPowerEventSuccess) ] ];
   // DCMicroGrid.Loads.Comm.Load05
   23: XIC(Load05DisconnectPowerInProcess)XIC(Load05DisconnectPowerEventSuccess)TON(Load05DisconnectPowerSuccessTimer,?,?);
   // DCMicroGrid.Loads.Comm.Load05
   24: XIC(Load05DisconnectPowerInProcess)XIC(Load05DisconnectPowerEventFail)TON(Load05DisconnectPowerFailTimer,?,?);
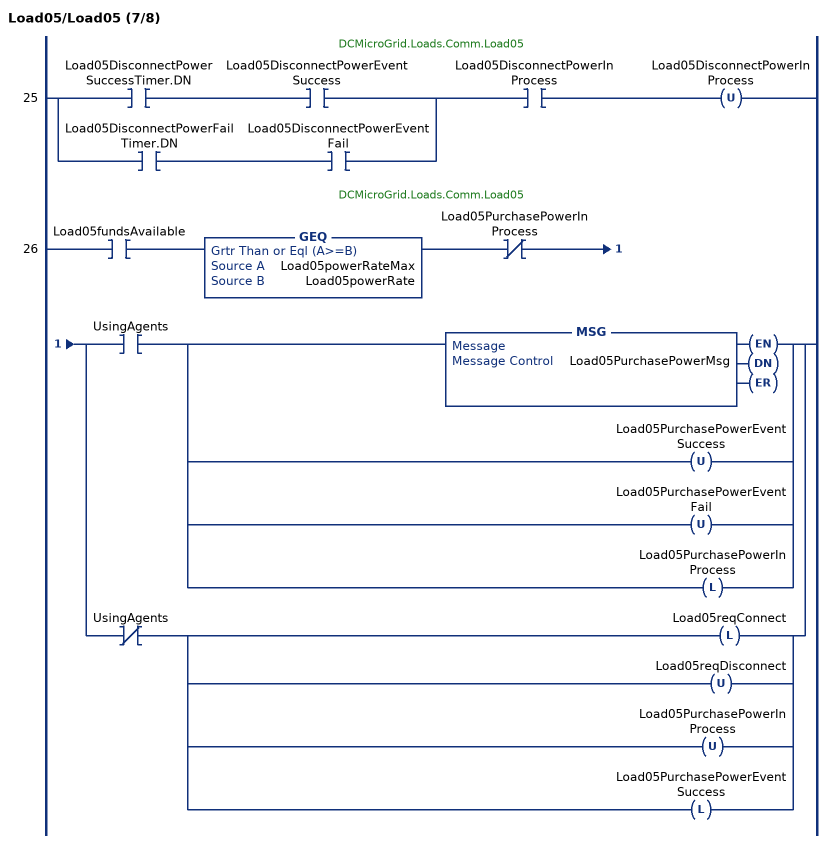
   // DCMicroGrid.Loads.Comm.Load05
   25: [XIC(Load05DisconnectPowerSuccessTimer.DN) XIC(Load05DisconnectPowerEventSuccess) ,XIC(Load05DisconnectPowerFailTimer.DN) XIC(Load05DisconnectPowerEventFail) ]XIC(Load05DisconnectPowerInProcess)OTU(Load05DisconnectPowerInProcess);
   // DCMicroGrid.Loads.Comm.Load05
   26: XIC(Load05fundsAvailable)GEQ(Load05powerRateMax,Load05powerRate)XIO(Load05PurchasePowerInProcess)[XIC(UsingAgents) [MSG(Load05PurchasePowerMsg) ,OTU(Load05PurchasePowerEventSuccess) ,OTU(Load05PurchasePowerEventFail) ,OTL(Load05PurchasePowerInProcess) ] ,XIO(UsingAgents) [OTL(Load05reqConnect) ,OTU(Load05reqDisconnect) ,OTU(Load05PurchasePowerInProcess) ,OTL(Load05PurchasePowerEventSuccess) ] ];
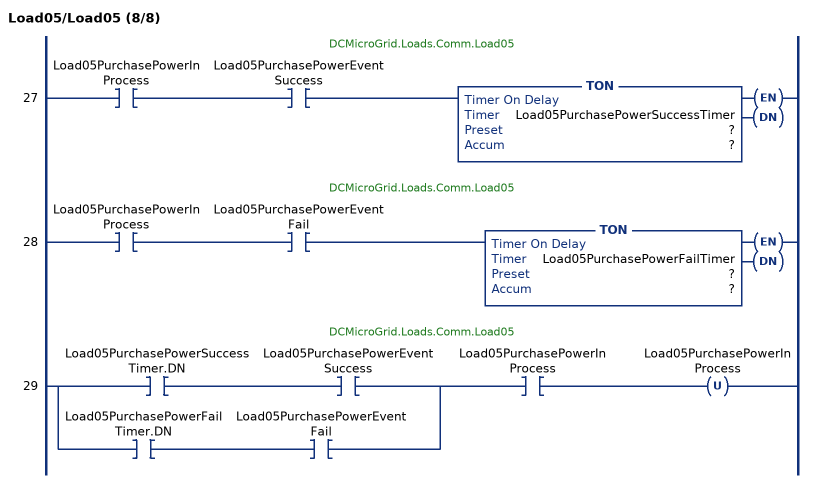
   // DCMicroGrid.Loads.Comm.Load05
   27: XIC(Load05PurchasePowerInProcess)XIC(Load05PurchasePowerEventSuccess)TON(Load05PurchasePowerSuccessTimer,?,?);
   // DCMicroGrid.Loads.Comm.Load05
   28: XIC(Load05PurchasePowerInProcess)XIC(Load05PurchasePowerEventFail)TON(Load05PurchasePowerFailTimer,?,?);
   // DCMicroGrid.Loads.Comm.Load05
   29: [XIC(Load05PurchasePowerSuccessTimer.DN) XIC(Load05PurchasePowerEventSuccess) ,XIC(Load05PurchasePowerFailTimer.DN) XIC(Load05PurchasePowerEventFail) ]XIC(Load05PurchasePowerInProcess)OTU(Load05PurchasePowerInProcess);
END_ROUTINE
END_PROGRAM
